Yaskawa INFORM job: R1_W30(0,0)OK-KM.JBI

/JOB
//NAME R1_W30(0,0)OK-KM
///FOLDERNAME SCIANA-NOWY-R2-KM
//POS
///NPOS 55,55,0,5,0,0
///TOOL 0
///POSTYPE PULSE
///PULSE
C00000=-14896,69737,-7372,13607,83025,-86522
C00001=-5831,-157881,-130818,18856,36102,-89754
C00002=117272,-157881,-130818,18856,4001,-90770
C00003=146352,-162940,-126965,-90343,92149,-37164
C00004=146352,-162940,-126965,-90343,92149,-37164
C00005=69533,-20928,-45802,-64911,81596,-45835
C00006=60350,-3569,-35626,-51441,69694,-41129
C00007=59024,1896,-26466,-51725,67182,-40340
C00008=58481,3234,-25331,-51504,66880,-40458
C00009=59024,1896,-26466,-51725,67182,-40340
C00010=59024,1681,-25597,-51932,66773,-40091
C00011=59024,1896,-26466,-51725,67182,-40340
C00012=56868,-6095,-33048,-50838,65992,-40800
C00013=56579,-3408,-26804,-51575,64255,-39911
C00014=56257,-2582,-26127,-51435,64084,-39989
C00015=56330,-2774,-26285,-51470,64124,-39971
C00016=56712,-843,-24690,-51622,64340,-39889
C00017=56579,-3408,-26804,-51575,64255,-39911
C00018=47968,-20086,-39698,-48020,59261,-41755
C00019=47867,-19912,-39857,-47891,59338,-41850
C00020=47413,-18545,-38854,-47635,59162,-42000
C00021=47441,-18629,-38918,-47654,59173,-41993
C00022=46832,-19549,-39593,-47384,58821,-42129
C00023=47867,-19912,-39857,-47891,59338,-41850
C00024=47867,-19316,-43044,-46954,60904,-42719
C00025=43801,-18075,-46073,-40418,64217,-45708
C00026=43503,-17060,-45320,-40250,64132,-45807
C00027=43801,-18075,-46073,-40418,64217,-45708
C00028=43801,-18293,-45436,-40574,63829,-45542
C00029=43801,-18075,-46073,-40418,64217,-45708
C00030=46029,-24455,-53452,-41167,66165,-45522
C00031=43606,-10551,-43125,-39698,71570,-40151
C00032=43897,-10172,-42685,-39843,71640,-40052
C00033=45629,-7482,-39959,-40666,72160,-39520
C00034=47000,-5950,-38385,-41294,72627,-39119
C00035=48354,-11837,-44148,-41773,73622,-38946
C00036=52499,-4356,-38225,-43942,76217,21975
C00037=57919,5325,-12872,-62013,76748,32701
C00038=58188,6092,-7535,-62643,75516,33948
C00039=59950,8546,-12220,-62246,78630,32522
C00040=36401,-38867,-50226,-3403,36055,1759
C00041=37842,-29016,-39166,-5272,34395,2678
C00042=37489,-28711,-37616,-4952,33576,2529
C00043=37404,-28742,-34327,-5129,31538,2626
C00044=35824,-35696,-44399,-2877,34081,1513
C00045=31819,-15527,-46431,6538,63892,51986
C00046=38354,-24308,-53392,-1518,53273,53160
C00047=47213,-1927,-40416,-14376,64099,60783
C00048=48826,3814,-34449,-18057,65902,63148
C00049=45819,-1765,-37916,-16379,64618,62276
C00050=45383,-10149,-44859,-16123,64502,62136
C00051=60301,-44333,-78630,-24159,70878,66236
C00052=146352,-162940,-126965,-90343,92149,-37164
C00053=146352,-162940,-126965,-90343,92149,-37164
C00054=17940,-162940,-126965,-1275,92149,-37164
BC00000=190810,830287,1069742
BC00001=366722,1154444,1065569
BC00002=24334,1154444,1065569
BC00003=876,1168099,1059656
BC00004=876,1168099,172418
BC00005=876,1168099,178053
BC00006=876,1164036,178053
BC00007=876,1164036,178053
BC00008=876,1164036,178053
BC00009=876,1164036,178053
BC00010=876,1164036,178053
BC00011=876,1164036,178053
BC00012=876,1164036,178053
BC00013=876,1161732,178053
BC00014=876,1161732,178053
BC00015=876,1161732,178053
BC00016=876,1161732,178053
BC00017=876,1161732,178053
BC00018=876,1161732,178053
BC00019=876,1161732,172676
BC00020=876,1161732,172676
BC00021=876,1161732,172676
BC00022=876,1161732,172676
BC00023=876,1161732,172676
BC00024=876,1161732,172676
BC00025=876,1164036,178053
BC00026=876,1164036,178053
BC00027=876,1164036,178053
BC00028=876,1164036,178053
BC00029=876,1164036,178053
BC00030=876,1164036,178053
BC00031=876,1164036,178053
BC00032=876,1164036,178053
BC00033=876,1164036,178053
BC00034=876,1164036,178051
BC00035=876,1164036,178051
BC00036=876,1164036,178049
BC00037=876,1164036,178049
BC00038=876,1164036,178049
BC00039=876,1164036,178049
BC00040=876,1164036,178049
BC00041=876,1164036,178049
BC00042=876,1164036,178049
BC00043=876,1164036,178049
BC00044=876,1164036,178049
BC00045=876,1164036,178049
BC00046=876,1164036,178049
BC00047=876,1164036,178048
BC00048=876,1164036,178047
BC00049=876,1164036,178047
BC00050=876,1164036,178047
BC00051=876,1164036,178047
BC00052=876,1168099,172418
BC00053=876,705782,1059656
BC00054=74742,705782,1059656
///POSTYPE BASE
///RECTAN
///RCONF 0,0,0,0,0,0,0,0,0,0,0,0,0,0,0,0,0,0,0,0,0,0,0,0
P00006=0.222,-3.123,-1.508,0.0000,0.0000,0.0000
P00022=0.222,-3.123,-1.508,0.0000,0.0000,0.0000
P00023=0.143,-0.036,0.682,0.0000,0.0000,0.0000
P00024=0.145,-0.552,1.326,0.0000,0.0000,0.0000
P00025=-2.003,0.006,0.728,0.0000,0.0000,0.0000
//INST
///DATE 2024/07/18 17:23
///ATTR SC,RW
///GROUP1 RB1,BS1
NOP
'r1_W30(0,0)
'Path VIA1137
SFTOF
MOVJ C00000 BC00000 VJ=100.00
MOVJ C00001 BC00001 VJ=50.00
MOVJ C00002 BC00002 VJ=50.00
MOVJ C00003 BC00003 VJ=100.00
'BRAK BLASZEK
MOVJ C00004 BC00004 VJ=100.00
MOVJ C00005 BC00005 VJ=50.00
MOVJ C00006 BC00006 VJ=50.00
MOVJ C00007 BC00007 VJ=15.00
REFP 3 C00008 BC00008
CALL JOB:SEARCH-R1
SET P022 P006
SFTON P022
MOVL C00009 BC00009 V=60.0
REFP 3 C00010 BC00010
CALL JOB:SEARCH-R1
SET P022 P006
SFTON P022
MOVL C00011 BC00011 V=60.0
SFTOF
MOVL C00012 BC00012 V=100.0
MOVL C00013 BC00013 V=100.0
REFP 3 C00014 BC00014
CALL JOB:SEARCH-R1
SET P023 P006
SFTON P023
MOVL C00015 BC00015 V=60.0
REFP 3 C00016 BC00016
CALL JOB:SEARCH-R1
SET P023 P006
SFTON P023
MOVL C00017 BC00017 V=60.0
SFTOF
MOVL C00018 BC00018 V=100.0
MOVL C00019 BC00019 V=100.0
REFP 3 C00020 BC00020
CALL JOB:SEARCH-R1
SET P025 P006
SFTON P025
MOVL C00021 BC00021 V=60.0
REFP 3 C00022 BC00022
CALL JOB:SEARCH-R1
SET P025 P006
SFTON P025
MOVL C00023 BC00023 V=60.0
MOVL C00024 BC00024 V=100.0
MOVL C00025 BC00025 V=100.0
REFP 3 C00026 BC00026
CALL JOB:SEARCH-R1
SET P024 P006
SFTON P024
MOVL C00027 BC00027 V=60.0
REFP 3 C00028 BC00028
CALL JOB:SEARCH-R1
SET P024 P006
SFTON P024
MOVL C00029 BC00029 V=60.0
MOVL C00030 BC00030 V=100.0
MACRO1 MJ#(0) ARGF7
SFTON P024
MOVL C00031 BC00031 V=100.0
ARCON
MOVL C00032 BC00032 V=10.0
MOVL C00033 BC00033 V=10.0
MOVL C00034 BC00034 V=10.0
ARCOF
MOVJ C00035 BC00035 VJ=15.00
SFTOF
MOVJ C00036 BC00036 VJ=15.00
SFTON P025
MOVL C00037 BC00037 V=83.3
ARCON
MOVL C00038 BC00038 V=11.7
ARCOF
MOVL C00039 BC00039 V=83.3
SFTOF
MOVL C00040 BC00040 V=83.3
SFTON P023
MOVL C00041 BC00041 V=83.3
ARCON
MOVL C00042 BC00042 V=11.7
MOVL C00043 BC00043 V=11.7
ARCOF
MOVJ C00044 BC00044 VJ=15.00
SFTOF
MOVJ C00045 BC00045 VJ=20.00
MOVJ C00046 BC00046 VJ=20.00
MOVJ C00047 BC00047 VJ=40.00
SFTON P022
MOVJ C00048 BC00048 VJ=20.00
ARCON
MOVL C00049 BC00049 V=10.0
ARCOF
MOVJ C00050 BC00050 VJ=20.00
SFTOF
MOVJ C00051 BC00051 VJ=40.00
MOVJ C00052 BC00052 VJ=40.00
MOVJ C00053 BC00053 VJ=100.00
MOVJ C00054 BC00054 VJ=70.00
END
